LIN {X 0,Y 72.884,Z 397.402,A -85,B 0,C 180,E1 -28001.113,E2 -28001.113} C_VEL
LIN {X 0,Y 72.584,Z 397.443,A -85,B 0,C 180,E1 -28006.88,E2 -28006.88} C_VEL
LIN {X 0,Y 72.397,Z 397.459,A -85,B 0,C 180,E1 -28012.842,E2 -28012.842} C_VEL
LIN {X 0,Y 72.372,Z 397.464,A -85,B 0,C 180,E1 -28019.077,E2 -28019.077} C_VEL
LIN {X 0,Y 72.344,Z 397.474,A -85,B 0,C 180,E1 -28025.645,E2 -28025.645} C_VEL
LIN {X 0,Y 72.326,Z 397.475,A -85,B 0,C 180,E1 -28032.85,E2 -28032.85} C_VEL
LIN {X 0,Y 72.365,Z 397.469,A -85,B 0,C 180,E1 -28040.971,E2 -28040.971} C_VEL
LIN {X 0,Y 72.342,Z 397.472,A -85,B 0,C 180,E1 -28044.346,E2 -28044.346} C_VEL
LIN {X 0,Y 72.385,Z 397.468,A -85,B 0,C 180,E1 -28050.958,E2 -28050.958} C_VEL
LIN {X 0,Y 72.392,Z 397.461,A -85,B 0,C 180,E1 -28057.15,E2 -28057.15} C_VEL
LIN {X 0,Y 72.749,Z 397.413,A -85,B 0,C 180,E1 -28065.002,E2 -28065.002} C_VEL
LIN {X 0,Y 72.877,Z 397.407,A -85,B 0,C 180,E1 -28068.88,E2 -28068.88} C_VEL
LIN {X 0,Y 73.573,Z 397.317,A -85,B 0,C 180,E1 -28080.001,E2 -28080.001} C_VEL
LIN {X 0,Y 72.877,Z 397.398,A -85,B 0,C 180,E1 -28091.121,E2 -28091.121} C_VEL
LIN {X 0,Y 72.575,Z 397.443,A -85,B 0,C 180,E1 -28096.889,E2 -28096.889} C_VEL
LIN {X 0,Y 72.388,Z 397.467,A -85,B 0,C 180,E1 -28102.853,E2 -28102.853} C_VEL
LIN {X 0,Y 72.37,Z 397.461,A -85,B 0,C 180,E1 -28109.086,E2 -28109.086} C_VEL
LIN {X 0,Y 72.341,Z 397.469,A -85,B 0,C 180,E1 -28115.656,E2 -28115.656} C_VEL
LIN {X 0,Y 72.336,Z 397.474,A -85,B 0,C 180,E1 -28122.853,E2 -28122.853} C_VEL
LIN {X 0,Y 72.557,Z 397.447,A -85,B 0,C 180,E1 -28130.797,E2 -28130.797} C_VEL
LIN {X 0,Y 73.99,Z 397.266,A -85,B 0,C 180,E1 -28141.653,E2 -28141.653} C_VEL
LIN {X 0,Y 75.709,Z 408.16,A -85,B 0,C 180,E1 -28143.6,E2 -28143.6} C_VEL
LIN {X 0,Y 76.943,Z 433.067,A -85,B 0,C 180,E1 -28148.277,E2 -28148.277} C_VEL
LIN {X 0,Y 79.549,Z 458.898,A -85,B 0,C 180,E1 -28152.824,E2 -28152.824} C_VEL
LIN {X 0,Y 80.052,Z 501.083,A -85,B 0,C 180,E1 -28161.567,E2 -28161.567} C_VEL
LIN {X 0,Y 80.299,Z 512.942,A -85,B 0,C 180,E1 -28164.985,E2 -28164.985} C_VEL
LIN {X 0,Y 80.965,Z 525.078,A -85,B 0,C 180,E1 -28169.384,E2 -28169.384} C_VEL
LIN {X 0,Y 82.181,Z 537.066,A -85,B 0,C 180,E1 -28174.911,E2 -28174.911} C_VEL
LIN {X 0,Y 83.655,Z 545.69,A -85,B 0,C 180,E1 -28179.678,E2 -28179.678} C_VEL
LIN {X 0,Y 84.498,Z 549.412,A -85,B 0,C 180,E1 -28182.007,E2 -28182.007} C_VEL
LIN {X 0,Y 84.134,Z 553.13,A -85,B 0,C 180,E1 -28186.037,E2 -28186.037} C_VEL
LIN {X 0,Y 85.067,Z 561.406,A -85,B 0,C 180,E1 -28197.032,E2 -28197.032} C_VEL
LIN {X 0,Y 89.087,Z 567.646,A -85,B 0,C 180,E1 -28206.277,E2 -28206.277} C_VEL
LIN {X 0,Y 97.647,Z 574.029,A -85,B 0,C 180,E1 -28216.039,E2 -28216.039} C_VEL
LIN {X 0,Y 97.752,Z 573.898,A -85,B 0,C 180,E1 -28217.096,E2 -28217.096} C_VEL
LIN {X 0,Y 89.651,Z 565.539,A -85,B 0,C 180,E1 -28223.988,E2 -28223.988} C_VEL
LIN {X 0,Y 83.684,Z 555.645,A -85,B 0,C 180,E1 -28232.489,E2 -28232.489} C_VEL
LIN {X 0,Y 80.707,Z 546.935,A -85,B 0,C 180,E1 -28239.615,E2 -28239.615} C_VEL
LIN {X 0,Y 78.9,Z 536.529,A -85,B 0,C 180,E1 -28247.133,E2 -28247.133} C_VEL
LIN {X 0,Y 78.177,Z 528.616,A -85,B 0,C 180,E1 -28251.99,E2 -28251.99} C_VEL
LIN {X 0,Y 77.712,Z 518.041,A -85,B 0,C 180,E1 -28257.408,E2 -28257.408} C_VEL
LIN {X 0,Y 77.597,Z 505.51,A -85,B 0,C 180,E1 -28262.595,E2 -28262.595} C_VEL
LIN {X 0,Y 77.899,Z 492.74,A -85,B 0,C 180,E1 -28266.748,E2 -28266.748} C_VEL
LIN {X 0,Y 78.228,Z 475.491,A -85,B 0,C 180,E1 -28270.841,E2 -28270.841} C_VEL
LIN {X 0,Y 78.384,Z 437.977,A -85,B 0,C 180,E1 -28278.458,E2 -28278.458} C_VEL
LIN {X 0,Y 78.852,Z 421.185,A -85,B 0,C 180,E1 -28281.786,E2 -28281.786} C_VEL
LIN {X 0,Y 78.146,Z 418.606,A -85,B 0,C 180,E1 -28282.165,E2 -28282.165} C_VEL
LIN {X 0,Y 76.516,Z 414.995,A -85,B 0,C 180,E1 -28282.614,E2 -28282.614} C_VEL
LIN {X 0,Y 68.201,Z 404.386,A -85,B 0,C 180,E1 -28283.502,E2 -28283.502} C_VEL
LIN {X 0,Y 66.794,Z 400.744,A -85,B 0,C 180,E1 -28284.067,E2 -28284.067} C_VEL
LIN {X 0,Y 66.334,Z 398.209,A -85,B 0,C 180,E1 -28284.613,E2 -28284.613} C_VEL
LIN {X 0,Y 65.413,Z 398.327,A -85,B 0,C 180,E1 -28292.493,E2 -28292.493} C_VEL
LIN {X 0,Y 65.189,Z 398.356,A -85,B 0,C 180,E1 -28300.994,E2 -28300.994} C_VEL
LIN {X 0,Y 65.209,Z 398.353,A -85,B 0,C 180,E1 -28309.701,E2 -28309.701} C_VEL
LIN {X 0,Y 65.258,Z 398.346,A -85,B 0,C 180,E1 -28319.491,E2 -28319.491} C_VEL
LIN {X 0,Y 65.242,Z 398.358,A -85,B 0,C 180,E1 -28324.469,E2 -28324.469} C_VEL
LIN {X 0,Y 65.627,Z 398.307,A -85,B 0,C 180,E1 -28334.536,E2 -28334.536} C_VEL
LIN {X 0,Y 65.757,Z 398.285,A -85,B 0,C 180,E1 -28337.65,E2 -28337.65} C_VEL
LIN {X 0,Y 66.495,Z 398.203,A -85,B 0,C 180,E1 -28349.993,E2 -28349.993} C_VEL
LIN {X 0,Y 65.782,Z 398.282,A -85,B 0,C 180,E1 -28362.33,E2 -28362.33} C_VEL
LIN {X 0,Y 65.388,Z 398.339,A -85,B 0,C 180,E1 -28368.803,E2 -28368.803} C_VEL
LIN {X 0,Y 65.247,Z 398.357,A -85,B 0,C 180,E1 -28375.514,E2 -28375.514} C_VEL
LIN {X 0,Y 65.215,Z 398.356,A -85,B 0,C 180,E1 -28382.595,E2 -28382.595} C_VEL
LIN {X 0,Y 65.26,Z 398.349,A -85,B 0,C 180,E1 -28391.076,E2 -28391.076} C_VEL
LIN {X 0,Y 65.276,Z 398.347,A -85,B 0,C 180,E1 -28399.76,E2 -28399.76} C_VEL
LIN {X 0,Y 65.254,Z 398.353,A -85,B 0,C 180,E1 -28409.483,E2 -28409.483} C_VEL
LIN {X 0,Y 65.241,Z 398.351,A -85,B 0,C 180,E1 -28414.476,E2 -28414.476} C_VEL
LIN {X 0,Y 65.644,Z 398.298,A -85,B 0,C 180,E1 -28424.458,E2 -28424.458} C_VEL
LIN {X 0,Y 65.775,Z 398.29,A -85,B 0,C 180,E1 -28427.662,E2 -28427.662} C_VEL
LIN {X 0,Y 66.497,Z 398.198,A -85,B 0,C 180,E1 -28440.001,E2 -28440.001} C_VEL
LIN {X 0,Y 65.768,Z 398.285,A -85,B 0,C 180,E1 -28452.341,E2 -28452.341} C_VEL
LIN {X 0,Y 65.378,Z 398.333,A -85,B 0,C 180,E1 -28458.815,E2 -28458.815} C_VEL
LIN {X 0,Y 65.24,Z 398.357,A -85,B 0,C 180,E1 -28465.525,E2 -28465.525} C_VEL
LIN {X 0,Y 65.213,Z 398.362,A -85,B 0,C 180,E1 -28472.606,E2 -28472.606} C_VEL
LIN {X 0,Y 65.266,Z 398.355,A -85,B 0,C 180,E1 -28481.093,E2 -28481.093} C_VEL
LIN {X 0,Y 65.441,Z 398.334,A -85,B 0,C 180,E1 -28489.891,E2 -28489.891} C_VEL
LIN {X 0,Y 67.071,Z 398.126,A -85,B 0,C 180,E1 -28502.682,E2 -28502.682} C_VEL
LIN {X 0,Y 68.779,Z 409.161,A -85,B 0,C 180,E1 -28504.855,E2 -28504.855} C_VEL
LIN {X 0,Y 70.255,Z 434.542,A -85,B 0,C 180,E1 -28510.085,E2 -28510.085} C_VEL
LIN {X 0,Y 72.876,Z 458.865,A -85,B 0,C 180,E1 -28514.729,E2 -28514.729} C_VEL
LIN {X 0,Y 73.916,Z 500.644,A -85,B 0,C 180,E1 -28524.208,E2 -28524.208} C_VEL
LIN {X 0,Y 74.379,Z 512.529,A -85,B 0,C 180,E1 -28527.976,E2 -28527.976} C_VEL
LIN {X 0,Y 75.35,Z 524.438,A -85,B 0,C 180,E1 -28532.679,E2 -28532.679} C_VEL
LIN {X 0,Y 76.78,Z 535.088,A -85,B 0,C 180,E1 -28537.898,E2 -28537.898} C_VEL
LIN {X 0,Y 78.569,Z 543.731,A -85,B 0,C 180,E1 -28542.928,E2 -28542.928} C_VEL
LIN {X 0,Y 79.079,Z 545.678,A -85,B 0,C 180,E1 -28544.152,E2 -28544.152} C_VEL
LIN {X 0,Y 79.134,Z 547.078,A -85,B 0,C 180,E1 -28545.458,E2 -28545.458} C_VEL
LIN {X 0,Y 79.462,Z 555.198,A -85,B 0,C 180,E1 -28556.252,E2 -28556.252} C_VEL
LIN {X 0,Y 83.073,Z 562.054,A -85,B 0,C 180,E1 -28566.32,E2 -28566.32} C_VEL
LIN {X 0,Y 89.595,Z 567.905,A -85,B 0,C 180,E1 -28575.091,E2 -28575.091} C_VEL
LIN {X 0,Y 89.992,Z 567.977,A -85,B 0,C 180,E1 -28576.643,E2 -28576.643} C_VEL
LIN {X 0,Y 81.965,Z 558.323,A -85,B 0,C 180,E1 -28584.635,E2 -28584.635} C_VEL
LIN {X 0,Y 77.144,Z 548.736,A -85,B 0,C 180,E1 -28592.901,E2 -28592.901} C_VEL
LIN {X 0,Y 74.209,Z 538.508,A -85,B 0,C 180,E1 -28600.929,E2 -28600.929} C_VEL
LIN {X 0,Y 72.923,Z 529.145,A -85,B 0,C 180,E1 -28607.475,E2 -28607.475} C_VEL
LIN {X 0,Y 71.984,Z 518.076,A -85,B 0,C 180,E1 -28613.693,E2 -28613.693} C_VEL
LIN {X 0,Y 71.557,Z 506.061,A -85,B 0,C 180,E1 -28619.165,E2 -28619.165} C_VEL
LIN {X 0,Y 71.591,Z 494.153,A -85,B 0,C 180,E1 -28623.517,E2 -28623.517} C_VEL
LIN {X 0,Y 71.771,Z 478.582,A -85,B 0,C 180,E1 -28627.737,E2 -28627.737} C_VEL
LIN {X 0,Y 71.636,Z 448.711,A -85,B 0,C 180,E1 -28634.56,E2 -28634.56} C_VEL
LIN {X 0,Y 71.869,Z 421.52,A -85,B 0,C 180,E1 -28640.517,E2 -28640.517} C_VEL
LIN {X 0,Y 67.195,Z 402.969,A -85,B 0,C 180,E1 -28643.639,E2 -28643.639} C_VEL
LIN {X 0,Y 66.794,Z 400.744,A -85,B 0,C 180,E1 -28644.067,E2 -28644.067} C_VEL
LIN {X 0,Y 66.151,Z 399.397,A -85,B 0,C 180,E1 -28644.879,E2 -28644.879} C_VEL
LIN {X 0,Y 64.817,Z 398.602,A -85,B 0,C 180,E1 -28646.815,E2 -28646.815} C_VEL
LIN {X 0,Y 60.938,Z 398.887,A -85,B 0,C 180,E1 -28654.521,E2 -28654.521} C_VEL
LIN {X 0,Y 58.572,Z 399.406,A -85,B 0,C 180,E1 -28663.21,E2 -28663.21} C_VEL
LIN {X 0,Y 58.022,Z 399.251,A -85,B 0,C 180,E1 -28672.443,E2 -28672.443} C_VEL
LIN {X 0,Y 58.163,Z 399.232,A -85,B 0,C 180,E1 -28677.76,E2 -28677.76} C_VEL
LIN {X 0,Y 58.155,Z 399.234,A -85,B 0,C 180,E1 -28681.083,E2 -28681.083} C_VEL
LIN {X 0,Y 58.519,Z 399.194,A -85,B 0,C 180,E1 -28693.899,E2 -28693.899} C_VEL
LIN {X 0,Y 58.802,Z 399.157,A -85,B 0,C 180,E1 -28703.128,E2 -28703.128} C_VEL
LIN {X 0,Y 59.386,Z 399.088,A -85,B 0,C 180,E1 -28709.992,E2 -28709.992} C_VEL
LIN {X 0,Y 58.824,Z 399.154,A -85,B 0,C 180,E1 -28716.854,E2 -28716.854} C_VEL
LIN {X 0,Y 58.535,Z 399.192,A -85,B 0,C 180,E1 -28726.157,E2 -28726.157} C_VEL
LIN {X 0,Y 58.155,Z 399.234,A -85,B 0,C 180,E1 -28738.898,E2 -28738.898} C_VEL
LIN {X 0,Y 58.08,Z 399.246,A -85,B 0,C 180,E1 -28747.221,E2 -28747.221} C_VEL
LIN {X 0,Y 58.102,Z 399.241,A -85,B 0,C 180,E1 -28756.519,E2 -28756.519} C_VEL
LIN {X 0,Y 58.078,Z 399.251,A -85,B 0,C 180,E1 -28762.769,E2 -28762.769} C_VEL
LIN {X 0,Y 58.152,Z 399.241,A -85,B 0,C 180,E1 -28771.091,E2 -28771.091} C_VEL
LIN {X 0,Y 58.53,Z 399.185,A -85,B 0,C 180,E1 -28783.834,E2 -28783.834} C_VEL
LIN {X 0,Y 58.816,Z 399.149,A -85,B 0,C 180,E1 -28793.138,E2 -28793.138} C_VEL
LIN {X 0,Y 59.389,Z 399.083,A -85,B 0,C 180,E1 -28800.001,E2 -28800.001} C_VEL
LIN {X 0,Y 58.816,Z 399.159,A -85,B 0,C 180,E1 -28806.864,E2 -28806.864} C_VEL
LIN {X 0,Y 58.518,Z 399.195,A -85,B 0,C 180,E1 -28816.128,E2 -28816.128} C_VEL
LIN {X 0,Y 58.15,Z 399.232,A -85,B 0,C 180,E1 -28828.911,E2 -28828.911} C_VEL
LIN {X 0,Y 58.081,Z 399.24,A -85,B 0,C 180,E1 -28837.231,E2 -28837.231} C_VEL
LIN {X 0,Y 58.186,Z 399.227,A -85,B 0,C 180,E1 -28846.446,E2 -28846.446} C_VEL
LIN {X 0,Y 58.897,Z 399.14,A -85,B 0,C 180,E1 -28856.648,E2 -28856.648} C_VEL
LIN {X 0,Y 60.22,Z 398.977,A -85,B 0,C 180,E1 -28864.088,E2 -28864.088} C_VEL
LIN {X 0,Y 61.903,Z 409.857,A -85,B 0,C 180,E1 -28866.433,E2 -28866.433} C_VEL
LIN {X 0,Y 63.446,Z 433.388,A -85,B 0,C 180,E1 -28871.799,E2 -28871.799} C_VEL
LIN {X 0,Y 66.355,Z 458.968,A -85,B 0,C 180,E1 -28877.137,E2 -28877.137} C_VEL
LIN {X 0,Y 68.011,Z 500.189,A -85,B 0,C 180,E1 -28887.416,E2 -28887.416} C_VEL
LIN {X 0,Y 68.741,Z 511.901,A -85,B 0,C 180,E1 -28891.471,E2 -28891.471} C_VEL
LIN {X 0,Y 70.075,Z 523.639,A -85,B 0,C 180,E1 -28896.485,E2 -28896.485} C_VEL
LIN {X 0,Y 72.148,Z 535.102,A -85,B 0,C 180,E1 -28902.523,E2 -28902.523} C_VEL
LIN {X 0,Y 73.814,Z 541.67,A -85,B 0,C 180,E1 -28906.603,E2 -28906.603} C_VEL
LIN {X 0,Y 74.056,Z 543.545,A -85,B 0,C 180,E1 -28908.372,E2 -28908.372} C_VEL
LIN {X 0,Y 75.288,Z 552.281,A -85,B 0,C 180,E1 -28920.557,E2 -28920.557} C_VEL
LIN {X 0,Y 80.097,Z 559.341,A -85,B 0,C 180,E1 -28931.16,E2 -28931.16} C_VEL
LIN {X 0,Y 82.912,Z 561.871,A -85,B 0,C 180,E1 -28934.893,E2 -28934.893} C_VEL
LIN {X 0,Y 81.955,Z 560.671,A -85,B 0,C 180,E1 -28936.682,E2 -28936.682} C_VEL
LIN {X 0,Y 74.644,Z 550.167,A -85,B 0,C 180,E1 -28945.602,E2 -28945.602} C_VEL
LIN {X 0,Y 70.806,Z 541.09,A -85,B 0,C 180,E1 -28953.306,E2 -28953.306} C_VEL
LIN {X 0,Y 68.092,Z 529.146,A -85,B 0,C 180,E1 -28962.428,E2 -28962.428} C_VEL
LIN {X 0,Y 66.732,Z 518.591,A -85,B 0,C 180,E1 -28968.995,E2 -28968.995} C_VEL
LIN {X 0,Y 65.901,Z 506.552,A -85,B 0,C 180,E1 -28975.065,E2 -28975.065} C_VEL
LIN {X 0,Y 65.609,Z 493.245,A -85,B 0,C 180,E1 -28980.383,E2 -28980.383} C_VEL
LIN {X 0,Y 65.57,Z 476.574,A -85,B 0,C 180,E1 -28985.284,E2 -28985.284} C_VEL
LIN {X 0,Y 64.904,Z 442.925,A -85,B 0,C 180,E1 -28993.731,E2 -28993.731} C_VEL
LIN {X 0,Y 65.039,Z 422.11,A -85,B 0,C 180,E1 -28998.813,E2 -28998.813} C_VEL
LIN {X 0,Y 60.331,Z 403.573,A -85,B 0,C 180,E1 -29002.159,E2 -29002.159} C_VEL
LIN {X 0,Y 59.457,Z 399.066,A -85,B 0,C 180,E1 -29003.193,E2 -29003.193} C_VEL
LIN {X 0,Y 58.104,Z 399.247,A -85,B 0,C 180,E1 -29017.212,E2 -29017.212} C_VEL
LIN {X 0,Y 58.018,Z 399.258,A -85,B 0,C 180,E1 -29026.618,E2 -29026.618} C_VEL
LIN {X 0,Y 58.022,Z 399.251,A -85,B 0,C 180,E1 -29032.443,E2 -29032.443} C_VEL
LIN {X 0,Y 57.853,Z 399.288,A -85,B 0,C 180,E1 -29036.305,E2 -29036.305} C_VEL
LIN {X 0,Y 56.621,Z 399.45,A -85,B 0,C 180,E1 -29042.093,E2 -29042.093} C_VEL
LIN {X 0,Y 54.829,Z 399.669,A -85,B 0,C 180,E1 -29047.958,E2 -29047.958} C_VEL
LIN {X 0,Y 51.867,Z 400.025,A -85,B 0,C 180,E1 -29061.019,E2 -29061.019} C_VEL
LIN {X 0,Y 51.817,Z 400.015,A -85,B 0,C 180,E1 -29065.612,E2 -29065.612} C_VEL
LIN {X 0,Y 52.269,Z 399.975,A -85,B 0,C 180,E1 -29069.991,E2 -29069.991} C_VEL
LIN {X 0,Y 51.7,Z 400.044,A -85,B 0,C 180,E1 -29077.804,E2 -29077.804} C_VEL
LIN {X 0,Y 51.401,Z 400.082,A -85,B 0,C 180,E1 -29086.847,E2 -29086.847} C_VEL
LIN {X 0,Y 51.027,Z 400.124,A -85,B 0,C 180,E1 -29094.395,E2 -29094.395} C_VEL
LIN {X 0,Y 51.053,Z 400.125,A -85,B 0,C 180,E1 -29104.315,E2 -29104.315} C_VEL
LIN {X 0,Y 51.067,Z 400.124,A -85,B 0,C 180,E1 -29113.468,E2 -29113.468} C_VEL
LIN {X 0,Y 51.067,Z 400.117,A -85,B 0,C 180,E1 -29116.52,E2 -29116.52} C_VEL
LIN {X 0,Y 51.074,Z 400.113,A -85,B 0,C 180,E1 -29126.605,E2 -29126.605} C_VEL
LIN {X 0,Y 51.023,Z 400.119,A -85,B 0,C 180,E1 -29135.593,E2 -29135.593} C_VEL
LIN {X 0,Y 51.474,Z 400.063,A -85,B 0,C 180,E1 -29144.154,E2 -29144.154} C_VEL
LIN {X 0,Y 51.692,Z 400.037,A -85,B 0,C 180,E1 -29152.187,E2 -29152.187} C_VEL
LIN {X 0,Y 52.274,Z 399.968,A -85,B 0,C 180,E1 -29160.001,E2 -29160.001} C_VEL
LIN {X 0,Y 51.69,Z 400.045,A -85,B 0,C 180,E1 -29167.815,E2 -29167.815} C_VEL
LIN {X 0,Y 51.386,Z 400.082,A -85,B 0,C 180,E1 -29176.822,E2 -29176.822} C_VEL
LIN {X 0,Y 51.021,Z 400.13,A -85,B 0,C 180,E1 -29184.409,E2 -29184.409} C_VEL
LIN {X 0,Y 51.052,Z 400.123,A -85,B 0,C 180,E1 -29194.329,E2 -29194.329} C_VEL
LIN {X 0,Y 51.168,Z 400.101,A -85,B 0,C 180,E1 -29206.639,E2 -29206.639} C_VEL
LIN {X 0,Y 52.619,Z 399.925,A -85,B 0,C 180,E1 -29222.144,E2 -29222.144} C_VEL
LIN {X 0,Y 53.445,Z 399.843,A -85,B 0,C 180,E1 -29226.07,E2 -29226.07} C_VEL
LIN {X 0,Y 55.057,Z 409.615,A -85,B 0,C 180,E1 -29228.28,E2 -29228.28} C_VEL
LIN {X 0,Y 57.04,Z 435.1,A -85,B 0,C 180,E1 -29234.716,E2 -29234.716} C_VEL
LIN {X 0,Y 60.017,Z 458.109,A -85,B 0,C 180,E1 -29239.891,E2 -29239.891} C_VEL
LIN {X 0,Y 62.423,Z 499.448,A -85,B 0,C 180,E1 -29251.218,E2 -29251.218} C_VEL
LIN {X 0,Y 63.485,Z 511.276,A -85,B 0,C 180,E1 -29255.647,E2 -29255.647} C_VEL
LIN {X 0,Y 64.967,Z 521.199,A -85,B 0,C 180,E1 -29260.132,E2 -29260.132} C_VEL
LIN {X 0,Y 67.209,Z 531.883,A -85,B 0,C 180,E1 -29265.937,E2 -29265.937} C_VEL
LIN {X 0,Y 69.019,Z 538.028,A -85,B 0,C 180,E1 -29269.767,E2 -29269.767} C_VEL
LIN {X 0,Y 69.27,Z 539.215,A -85,B 0,C 180,E1 -29270.828,E2 -29270.828} C_VEL
LIN {X 0,Y 71.033,Z 547.999,A -85,B 0,C 180,E1 -29283.485,E2 -29283.485} C_VEL
LIN {X 0,Y 76.015,Z 554.814,A -85,B 0,C 180,E1 -29293.837,E2 -29293.837} C_VEL
LIN {X 0,Y 75.472,Z 553.984,A -85,B 0,C 180,E1 -29295.7,E2 -29295.7} C_VEL
LIN {X 0,Y 68.382,Z 542.524,A -85,B 0,C 180,E1 -29305.575,E2 -29305.575} C_VEL
LIN {X 0,Y 64.548,Z 532.018,A -85,B 0,C 180,E1 -29314.181,E2 -29314.181} C_VEL
LIN {X 0,Y 62.84,Z 523.725,A -85,B 0,C 180,E1 -29320.395,E2 -29320.395} C_VEL
LIN {X 0,Y 61.304,Z 513.354,A -85,B 0,C 180,E1 -29326.744,E2 -29326.744} C_VEL
LIN {X 0,Y 60.319,Z 502.043,A -85,B 0,C 180,E1 -29332.467,E2 -29332.467} C_VEL
LIN {X 0,Y 59.891,Z 489.793,A -85,B 0,C 180,E1 -29337.477,E2 -29337.477} C_VEL
LIN {X 0,Y 59.468,Z 472.762,A -85,B 0,C 180,E1 -29342.751,E2 -29342.751} C_VEL
LIN {X 0,Y 58.275,Z 438.279,A -85,B 0,C 180,E1 -29352.297,E2 -29352.297} C_VEL
LIN {X 0,Y 58.235,Z 422.432,A -85,B 0,C 180,E1 -29356.652,E2 -29356.652} C_VEL
LIN {X 0,Y 53.572,Z 404.309,A -85,B 0,C 180,E1 -29360.124,E2 -29360.124} C_VEL
LIN {X 0,Y 52.653,Z 399.921,A -85,B 0,C 180,E1 -29361.338,E2 -29361.338} C_VEL
LIN {X 0,Y 51.143,Z 400.106,A -85,B 0,C 180,E1 -29374.446,E2 -29374.446} C_VEL
LIN {X 0,Y 50.985,Z 400.134,A -85,B 0,C 180,E1 -29386.419,E2 -29386.419} C_VEL
LIN {X 0,Y 51.055,Z 400.122,A -85,B 0,C 180,E1 -29396.58,E2 -29396.58} C_VEL
LIN {X 0,Y 51.026,Z 400.125,A -85,B 0,C 180,E1 -29405.584,E2 -29405.584} C_VEL
LIN {X 0,Y 51.46,Z 400.072,A -85,B 0,C 180,E1 -29414.139,E2 -29414.139} C_VEL
LIN {X 0,Y 51.817,Z 400.015,A -85,B 0,C 180,E1 -29425.612,E2 -29425.612} C_VEL
LIN {X 0,Y 51.492,Z 400.071,A -85,B 0,C 180,E1 -29429.149,E2 -29429.149} C_VEL
LIN {X 0,Y 49.798,Z 400.291,A -85,B 0,C 180,E1 -29433.965,E2 -29433.965} C_VEL
LIN {X 0,Y 44.332,Z 400.965,A -85,B 0,C 180,E1 -29447.752,E2 -29447.752} C_VEL
LIN {X 0,Y 44.096,Z 400.983,A -85,B 0,C 180,E1 -29449.551,E2 -29449.551} C_VEL
LIN {X 0,Y 43.856,Z 401.015,A -85,B 0,C 180,E1 -29458.722,E2 -29458.722} C_VEL
LIN {X 0,Y 43.873,Z 401.01,A -85,B 0,C 180,E1 -29469.835,E2 -29469.835} C_VEL
LIN {X 0,Y 43.907,Z 401.016,A -85,B 0,C 180,E1 -29483.142,E2 -29483.142} C_VEL
LIN {X 0,Y 43.853,Z 401.023,A -85,B 0,C 180,E1 -29491.264,E2 -29491.264} C_VEL
LIN {X 0,Y 44.25,Z 400.967,A -85,B 0,C 180,E1 -29502.317,E2 -29502.317} C_VEL
LIN {X 0,Y 44.544,Z 400.931,A -85,B 0,C 180,E1 -29510.923,E2 -29510.923} C_VEL
LIN {X 0,Y 45.149,Z 400.855,A -85,B 0,C 180,E1 -29520.001,E2 -29520.001} C_VEL
LIN {X 0,Y 44.539,Z 400.93,A -85,B 0,C 180,E1 -29529.08,E2 -29529.08} C_VEL
LIN {X 0,Y 44.15,Z 400.976,A -85,B 0,C 180,E1 -29538.566,E2 -29538.566} C_VEL
LIN {X 0,Y 43.853,Z 401.012,A -85,B 0,C 180,E1 -29548.738,E2 -29548.738} C_VEL
LIN {X 0,Y 43.896,Z 401.012,A -85,B 0,C 180,E1 -29559.825,E2 -29559.825} C_VEL
LIN {X 0,Y 44.308,Z 400.96,A -85,B 0,C 180,E1 -29572.477,E2 -29572.477} C_VEL
LIN {X 0,Y 46.765,Z 400.659,A -85,B 0,C 180,E1 -29588.607,E2 -29588.607} C_VEL
LIN {X 0,Y 48.333,Z 409.803,A -85,B 0,C 180,E1 -29590.958,E2 -29590.958} C_VEL
LIN {X 0,Y 50.773,Z 435.813,A -85,B 0,C 180,E1 -29598.24,E2 -29598.24} C_VEL
LIN {X 0,Y 53.923,Z 458.116,A -85,B 0,C 180,E1 -29603.695,E2 -29603.695} C_VEL
LIN {X 0,Y 57.212,Z 498.454,A -85,B 0,C 180,E1 -29615.735,E2 -29615.735} C_VEL
LIN {X 0,Y 58.633,Z 510.019,A -85,B 0,C 180,E1 -29620.366,E2 -29620.366} C_VEL
LIN {X 0,Y 60.601,Z 520.498,A -85,B 0,C 180,E1 -29625.396,E2 -29625.396} C_VEL
LIN {X 0,Y 63.706,Z 531.833,A -85,B 0,C 180,E1 -29631.885,E2 -29631.885} C_VEL
LIN {X 0,Y 64.779,Z 534.938,A -85,B 0,C 180,E1 -29633.908,E2 -29633.908} C_VEL
LIN {X 0,Y 67.404,Z 544.014,A -85,B 0,C 180,E1 -29647.44,E2 -29647.44} C_VEL
LIN {X 0,Y 69.896,Z 547.579,A -85,B 0,C 180,E1 -29652.96,E2 -29652.96} C_VEL
LIN {X 0,Y 69.317,Z 546.679,A -85,B 0,C 180,E1 -29654.786,E2 -29654.786} C_VEL
LIN {X 0,Y 63.264,Z 536.075,A -85,B 0,C 180,E1 -29663.846,E2 -29663.846} C_VEL
LIN {X 0,Y 59.175,Z 524.061,A -85,B 0,C 180,E1 -29673.552,E2 -29673.552} C_VEL
LIN {X 0,Y 57.094,Z 514.187,A -85,B 0,C 180,E1 -29680.213,E2 -29680.213} C_VEL
LIN {X 0,Y 55.612,Z 503.425,A -85,B 0,C 180,E1 -29686.292,E2 -29686.292} C_VEL
LIN {X 0,Y 54.634,Z 490.582,A -85,B 0,C 180,E1 -29692.144,E2 -29692.144} C_VEL
LIN {X 0,Y 53.818,Z 473.473,A -85,B 0,C 180,E1 -29698.128,E2 -29698.128} C_VEL
LIN {X 0,Y 52.002,Z 440.349,A -85,B 0,C 180,E1 -29708.347,E2 -29708.347} C_VEL
LIN {X 0,Y 51.519,Z 422.361,A -85,B 0,C 180,E1 -29713.897,E2 -29713.897} C_VEL
LIN {X 0,Y 46.851,Z 404.631,A -85,B 0,C 180,E1 -29717.457,E2 -29717.457} C_VEL
LIN {X 0,Y 46.049,Z 400.748,A -85,B 0,C 180,E1 -29718.505,E2 -29718.505} C_VEL
LIN {X 0,Y 43.932,Z 401.013,A -85,B 0,C 180,E1 -29736.865,E2 -29736.865} C_VEL
LIN {X 0,Y 43.806,Z 401.018,A -85,B 0,C 180,E1 -29750.065,E2 -29750.065} C_VEL
LIN {X 0,Y 43.847,Z 401.016,A -85,B 0,C 180,E1 -29761.247,E2 -29761.247} C_VEL
LIN {X 0,Y 44.231,Z 400.976,A -85,B 0,C 180,E1 -29772.43,E2 -29772.43} C_VEL
LIN {X 0,Y 44.531,Z 400.938,A -85,B 0,C 180,E1 -29780.909,E2 -29780.909} C_VEL
LIN {X 0,Y 45.143,Z 400.862,A -85,B 0,C 180,E1 -29789.99,E2 -29789.99} C_VEL
LIN {X 0,Y 44.551,Z 400.936,A -85,B 0,C 180,E1 -29799.066,E2 -29799.066} C_VEL
LIN {X 0,Y 44.096,Z 400.983,A -85,B 0,C 180,E1 -29809.551,E2 -29809.551} C_VEL
LIN {X 0,Y 43.388,Z 401.076,A -85,B 0,C 180,E1 -29814.623,E2 -29814.623} C_VEL
LIN {X 0,Y 41.673,Z 401.291,A -85,B 0,C 180,E1 -29822.278,E2 -29822.278} C_VEL
LIN {X 0,Y 39.664,Z 401.534,A -85,B 0,C 180,E1 -29830.224,E2 -29830.224} C_VEL
LIN {X 0,Y 36.682,Z 401.889,A -85,B 0,C 180,E1 -29854.884,E2 -29854.884} C_VEL
LIN {X 0,Y 37.074,Z 401.864,A -85,B 0,C 180,E1 -29861.37,E2 -29861.37} C_VEL
LIN {X 0,Y 37.342,Z 401.834,A -85,B 0,C 180,E1 -29869.153,E2 -29869.153} C_VEL
LIN {X 0,Y 38.007,Z 401.743,A -85,B 0,C 180,E1 -29880.001,E2 -29880.001} C_VEL
LIN {X 0,Y 37.331,Z 401.824,A -85,B 0,C 180,E1 -29890.853,E2 -29890.853} C_VEL
LIN {X 0,Y 37.052,Z 401.86,A -85,B 0,C 180,E1 -29898.527,E2 -29898.527} C_VEL
LIN {X 0,Y 36.757,Z 401.899,A -85,B 0,C 180,E1 -29915.003,E2 -29915.003} C_VEL
LIN {X 0,Y 36.836,Z 401.892,A -85,B 0,C 180,E1 -29920.275,E2 -29920.275} C_VEL
LIN {X 0,Y 37.44,Z 401.811,A -85,B 0,C 180,E1 -29935.743,E2 -29935.743} C_VEL
LIN {X 0,Y 40.252,Z 401.461,A -85,B 0,C 180,E1 -29952.141,E2 -29952.141} C_VEL
LIN {X 0,Y 41.826,Z 409.981,A -85,B 0,C 180,E1 -29954.619,E2 -29954.619} C_VEL
LIN {X 0,Y 44.866,Z 436.866,A -85,B 0,C 180,E1 -29962.981,E2 -29962.981} C_VEL
LIN {X 0,Y 48.206,Z 457.818,A -85,B 0,C 180,E1 -29968.443,E2 -29968.443} C_VEL
LIN {X 0,Y 52.403,Z 496.818,A -85,B 0,C 180,E1 -29980.969,E2 -29980.969} C_VEL
LIN {X 0,Y 53.969,Z 506.894,A -85,B 0,C 180,E1 -29985.105,E2 -29985.105} C_VEL
LIN {X 0,Y 56.657,Z 518.761,A -85,B 0,C 180,E1 -29990.902,E2 -29990.902} C_VEL
LIN {X 0,Y 60.035,Z 529.169,A -85,B 0,C 180,E1 -29996.926,E2 -29996.926} C_VEL
LIN {X 0,Y 60.488,Z 530.385,A -85,B 0,C 180,E1 -29997.703,E2 -29997.703} C_VEL
LIN {X 0,Y 60.902,Z 531.883,A -85,B 0,C 180,E1 -29999.38,E2 -29999.38} C_VEL
LIN {X 0,Y 63.997,Z 539.515,A -85,B 0,C 180,E1 -30011.226,E2 -30011.226} C_VEL
LIN {X 0,Y 62.912,Z 537.776,A -85,B 0,C 180,E1 -30014.564,E2 -30014.564} C_VEL
LIN {X 0,Y 58.747,Z 529.93,A -85,B 0,C 180,E1 -30021.089,E2 -30021.089} C_VEL
LIN {X 0,Y 55.091,Z 519.736,A -85,B 0,C 180,E1 -30029.316,E2 -30029.316} C_VEL
LIN {X 0,Y 52.517,Z 509.133,A -85,B 0,C 180,E1 -30036.329,E2 -30036.329} C_VEL
LIN {X 0,Y 50.652,Z 497.279,A -85,B 0,C 180,E1 -30042.851,E2 -30042.851} C_VEL
LIN {X 0,Y 49.518,Z 484.586,A -85,B 0,C 180,E1 -30048.486,E2 -30048.486} C_VEL
LIN {X 0,Y 47.903,Z 465.058,A -85,B 0,C 180,E1 -30055.529,E2 -30055.529} C_VEL
LIN {X 0,Y 45.18,Z 422.904,A -85,B 0,C 180,E1 -30070.08,E2 -30070.08} C_VEL
LIN {X 0,Y 40.651,Z 406.325,A -85,B 0,C 180,E1 -30073.429,E2 -30073.429} C_VEL
LIN {X 0,Y 39.554,Z 401.548,A -85,B 0,C 180,E1 -30074.862,E2 -30074.862} C_VEL
LIN {X 0,Y 36.923,Z 401.877,A -85,B 0,C 180,E1 -30094.82,E2 -30094.82} C_VEL
LIN {X 0,Y 36.769,Z 401.896,A -85,B 0,C 180,E1 -30100.114,E2 -30100.114} C_VEL
LIN {X 0,Y 36.732,Z 401.899,A -85,B 0,C 180,E1 -30109.935,E2 -30109.935} C_VEL
LIN {X 0,Y 36.727,Z 401.911,A -85,B 0,C 180,E1 -30114.95,E2 -30114.95} C_VEL
LIN {X 0,Y 37.057,Z 401.866,A -85,B 0,C 180,E1 -30131.485,E2 -30131.485} C_VEL
LIN {X 0,Y 37.329,Z 401.828,A -85,B 0,C 180,E1 -30139.135,E2 -30139.135} C_VEL
LIN {X 0,Y 38.001,Z 401.752,A -85,B 0,C 180,E1 -30149.988,E2 -30149.988} C_VEL
LIN {X 0,Y 37.348,Z 401.826,A -85,B 0,C 180,E1 -30160.833,E2 -30160.833} C_VEL
LIN {X 0,Y 37.079,Z 401.863,A -85,B 0,C 180,E1 -30168.616,E2 -30168.616} C_VEL
LIN {X 0,Y 36.757,Z 401.907,A -85,B 0,C 180,E1 -30184.986,E2 -30184.986} C_VEL
LIN {X 0,Y 36.782,Z 401.893,A -85,B 0,C 180,E1 -30190.158,E2 -30190.158} C_VEL
LIN {X 0,Y 36.781,Z 401.894,A -85,B 0,C 180,E1 -30199.826,E2 -30199.826} C_VEL
LIN {X 0,Y 36.765,Z 401.898,A -85,B 0,C 180,E1 -30205.008,E2 -30205.008} C_VEL
LIN {X 0,Y 36.682,Z 401.889,A -85,B 0,C 180,E1 -30214.884,E2 -30214.884} C_VEL
LIN {X 0,Y 36.394,Z 401.952,A -85,B 0,C 180,E1 -30219.899,E2 -30219.899} C_VEL
LIN {X 0,Y 34.873,Z 402.146,A -85,B 0,C 180,E1 -30226.856,E2 -30226.856} C_VEL
LIN {X 0,Y 30.12,Z 402.6,A -85,B 0,C 180,E1 -30250.355,E2 -30250.355} C_VEL
LIN {X 0,Y 29.869,Z 402.635,A -85,B 0,C 180,E1 -30259.797,E2 -30259.797} C_VEL
LIN {X 0,Y 29.545,Z 402.666,A -85,B 0,C 180,E1 -30268.409,E2 -30268.409} C_VEL
LIN {X 0,Y 29.768,Z 402.646,A -85,B 0,C 180,E1 -30285.097,E2 -30285.097} C_VEL
LIN {X 0,Y 32.449,Z 402.393,A -85,B 0,C 180,E1 -30311.057,E2 -30311.057} C_VEL
LIN {X 0,Y 34.097,Z 402.432,A -85,B 0,C 180,E1 -30317.449,E2 -30317.449} C_VEL
LIN {X 0,Y 35.664,Z 410.432,A -85,B 0,C 180,E1 -30319.845,E2 -30319.845} C_VEL
LIN {X 0,Y 38.977,Z 435.166,A -85,B 0,C 180,E1 -30328.398,E2 -30328.398} C_VEL
LIN {X 0,Y 42.952,Z 457.162,A -85,B 0,C 180,E1 -30334.391,E2 -30334.391} C_VEL
LIN {X 0,Y 48.578,Z 497.018,A -85,B 0,C 180,E1 -30347.915,E2 -30347.915} C_VEL
LIN {X 0,Y 51.164,Z 509.167,A -85,B 0,C 180,E1 -30353.27,E2 -30353.27} C_VEL
LIN {X 0,Y 54.467,Z 520.136,A -85,B 0,C 180,E1 -30358.948,E2 -30358.948} C_VEL
LIN {X 0,Y 56.972,Z 526.471,A -85,B 0,C 180,E1 -30362.614,E2 -30362.614} C_VEL
LIN {X 0,Y 57.312,Z 527.337,A -85,B 0,C 180,E1 -30363.423,E2 -30363.423} C_VEL
LIN {X 0,Y 58.698,Z 531.027,A -85,B 0,C 180,E1 -30369.329,E2 -30369.329} C_VEL
LIN {X 0,Y 58.784,Z 531.304,A -85,B 0,C 180,E1 -30371.648,E2 -30371.648} C_VEL
LIN {X 0,Y 53.064,Z 519.625,A -85,B 0,C 180,E1 -30381.014,E2 -30381.014} C_VEL
LIN {X 0,Y 50.606,Z 512.35,A -85,B 0,C 180,E1 -30386.253,E2 -30386.253} C_VEL
LIN {X 0,Y 48.001,Z 501.953,A -85,B 0,C 180,E1 -30392.652,E2 -30392.652} C_VEL
LIN {X 0,Y 45.861,Z 488.552,A -85,B 0,C 180,E1 -30399.537,E2 -30399.537} C_VEL
LIN {X 0,Y 43.84,Z 471.564,A -85,B 0,C 180,E1 -30406.414,E2 -30406.414} C_VEL
LIN {X 0,Y 40.05,Z 437.012,A -85,B 0,C 180,E1 -30419.37,E2 -30419.37} C_VEL
LIN {X 0,Y 38.997,Z 422.936,A -85,B 0,C 180,E1 -30424.957,E2 -30424.957} C_VEL
LIN {X 0,Y 34.341,Z 406.278,A -85,B 0,C 180,E1 -30428.265,E2 -30428.265} C_VEL
LIN {X 0,Y 33.349,Z 402.311,A -85,B 0,C 180,E1 -30429.563,E2 -30429.563} C_VEL
LIN {X 0,Y 30.23,Z 402.606,A -85,B 0,C 180,E1 -30447.706,E2 -30447.706} C_VEL
LIN {X 0,Y 29.586,Z 402.666,A -85,B 0,C 180,E1 -30465.448,E2 -30465.448} C_VEL
LIN {X 0,Y 29.498,Z 402.672,A -85,B 0,C 180,E1 -30481.525,E2 -30481.525} C_VEL
LIN {X 0,Y 29.866,Z 402.638,A -85,B 0,C 180,E1 -30490.263,E2 -30490.263} C_VEL
LIN {X 0,Y 30.107,Z 402.614,A -85,B 0,C 180,E1 -30496.485,E2 -30496.485} C_VEL
LIN {X 0,Y 30.818,Z 402.551,A -85,B 0,C 180,E1 -30509.985,E2 -30509.985} C_VEL
LIN {X 0,Y 30.126,Z 402.612,A -85,B 0,C 180,E1 -30523.475,E2 -30523.475} C_VEL
LIN {X 0,Y 29.89,Z 402.635,A -85,B 0,C 180,E1 -30529.867,E2 -30529.867} C_VEL
LIN {X 0,Y 29.554,Z 402.667,A -85,B 0,C 180,E1 -30538.381,E2 -30538.381} C_VEL
LIN {X 0,Y 29.596,Z 402.664,A -85,B 0,C 180,E1 -30555.406,E2 -30555.406} C_VEL
LIN {X 0,Y 29.555,Z 402.668,A -85,B 0,C 180,E1 -30571.604,E2 -30571.604} C_VEL
LIN {X 0,Y 29.885,Z 402.637,A -85,B 0,C 180,E1 -30580.115,E2 -30580.115} C_VEL
LIN {X 0,Y 30.12,Z 402.613,A -85,B 0,C 180,E1 -30586.508,E2 -30586.508} C_VEL
LIN {X 0,Y 30.824,Z 402.547,A -85,B 0,C 180,E1 -30600.001,E2 -30600.001} C_VEL
LIN {X 0,Y 30.12,Z 402.6,A -85,B 0,C 180,E1 -30610.355,E2 -30610.355} C_VEL
LIN {X 0,Y 29.579,Z 402.665,A -85,B 0,C 180,E1 -30617.683,E2 -30617.683} C_VEL
LIN {X 0,Y 28.201,Z 402.794,A -85,B 0,C 180,E1 -30626.968,E2 -30626.968} C_VEL
LIN {X 0,Y 25.96,Z 402.967,A -85,B 0,C 180,E1 -30640.966,E2 -30640.966} C_VEL
LIN {X 0,Y 25.576,Z 402.979,A -85,B 0,C 180,E1 -30674.481,E2 -30674.481} C_VEL
LIN {X 0,Y 26.456,Z 402.905,A -85,B 0,C 180,E1 -30678.723,E2 -30678.723} C_VEL
LIN {X 0,Y 28.231,Z 402.791,A -85,B 0,C 180,E1 -30684.761,E2 -30684.761} C_VEL
LIN {X 0,Y 29.958,Z 410.723,A -85,B 0,C 180,E1 -30687.291,E2 -30687.291} C_VEL
LIN {X 0,Y 34.388,Z 437.273,A -85,B 0,C 180,E1 -30696.933,E2 -30696.933} C_VEL
LIN {X 0,Y 38.464,Z 457.09,A -85,B 0,C 180,E1 -30702.209,E2 -30702.209} C_VEL
LIN {X 0,Y 45.533,Z 496.535,A -85,B 0,C 180,E1 -30715.74,E2 -30715.74} C_VEL
LIN {X 0,Y 48.963,Z 509.329,A -85,B 0,C 180,E1 -30721.365,E2 -30721.365} C_VEL
LIN {X 0,Y 52.866,Z 519.825,A -85,B 0,C 180,E1 -30726.738,E2 -30726.738} C_VEL
LIN {X 0,Y 54.16,Z 522.665,A -85,B 0,C 180,E1 -30728.292,E2 -30728.292} C_VEL
LIN {X 0,Y 54.391,Z 523.256,A -85,B 0,C 180,E1 -30729.169,E2 -30729.169} C_VEL
LIN {X 0,Y 49.788,Z 513.707,A -85,B 0,C 180,E1 -30736.515,E2 -30736.515} C_VEL
LIN {X 0,Y 46.044,Z 502.644,A -85,B 0,C 180,E1 -30743.48,E2 -30743.48} C_VEL
LIN {X 0,Y 42.991,Z 489.127,A -85,B 0,C 180,E1 -30750.63,E2 -30750.63} C_VEL
LIN {X 0,Y 40.582,Z 474.523,A -85,B 0,C 180,E1 -30756.855,E2 -30756.855} C_VEL
LIN {X 0,Y 36.933,Z 451.494,A -85,B 0,C 180,E1 -30765.78,E2 -30765.78} C_VEL
LIN {X 0,Y 33.414,Z 423.149,A -85,B 0,C 180,E1 -30777.795,E2 -30777.795} C_VEL
LIN {X 0,Y 28.408,Z 405.786,A -85,B 0,C 180,E1 -30780.826,E2 -30780.826} C_VEL
LIN {X 0,Y 27.602,Z 402.849,A -85,B 0,C 180,E1 -30781.759,E2 -30781.759} C_VEL
LIN {X 0,Y 23.253,Z 403.051,A -85,B 0,C 180,E1 -30804.895,E2 -30804.895} C_VEL
LIN {X 0,Y 22.423,Z 403.077,A -85,B 0,C 180,E1 -30818.817,E2 -30818.817} C_VEL
LIN {X 0,Y 22.218,Z 403.084,A -85,B 0,C 180,E1 -30830.728,E2 -30830.728} C_VEL
LIN {X 0,Y 22.813,Z 403.065,A -85,B 0,C 180,E1 -30852.036,E2 -30852.036} C_VEL
LIN {X 0,Y 23.587,Z 403.042,A -85,B 0,C 180,E1 -30869.98,E2 -30869.98} C_VEL
LIN {X 0,Y 22.842,Z 403.064,A -85,B 0,C 180,E1 -30887.898,E2 -30887.898} C_VEL
LIN {X 0,Y 22.236,Z 403.083,A -85,B 0,C 180,E1 -30909.179,E2 -30909.179} C_VEL
LIN {X 0,Y 22.236,Z 403.083,A -85,B 0,C 180,E1 -30920.796,E2 -30920.796} C_VEL
LIN {X 0,Y 22.837,Z 403.064,A -85,B 0,C 180,E1 -30942.079,E2 -30942.079} C_VEL
LIN {X 0,Y 23.591,Z 403.042,A -85,B 0,C 180,E1 -30960.002,E2 -30960.002} C_VEL
LIN {X 0,Y 22.821,Z 403.065,A -85,B 0,C 180,E1 -30977.939,E2 -30977.939} C_VEL
LIN {X 0,Y 22.311,Z 403.081,A -85,B 0,C 180,E1 -30999.053,E2 -30999.053} C_VEL
LIN {X 0,Y 22.786,Z 403.066,A -85,B 0,C 180,E1 -31011.939,E2 -31011.939} C_VEL
LIN {X 0,Y 26.456,Z 402.905,A -85,B 0,C 180,E1 -31038.723,E2 -31038.723} C_VEL
LIN {X 0,Y 26.989,Z 403.378,A -85,B 0,C 180,E1 -31042.756,E2 -31042.756} C_VEL
LIN {X 0,Y 26.737,Z 405.4,A -85,B 0,C 180,E1 -31048.707,E2 -31048.707} C_VEL
LIN {X 0,Y 25.427,Z 410.485,A -85,B 0,C 180,E1 -31056.631,E2 -31056.631} C_VEL
LIN {X 0,Y 25.297,Z 414.36,A -85,B 0,C 180,E1 -31060.5,E2 -31060.5} C_VEL
LIN {X 0,Y 26.091,Z 420.031,A -85,B 0,C 180,E1 -31063.257,E2 -31063.257} C_VEL
LIN {X 0,Y 29.092,Z 431.47,A -85,B 0,C 180,E1 -31065.785,E2 -31065.785} C_VEL
LIN {X 0,Y 34.906,Z 456.661,A -85,B 0,C 180,E1 -31071.805,E2 -31071.805} C_VEL
LIN {X 0,Y 43.223,Z 494.792,A -85,B 0,C 180,E1 -31084.135,E2 -31084.135} C_VEL
LIN {X 0,Y 46.972,Z 506.892,A -85,B 0,C 180,E1 -31089.005,E2 -31089.005} C_VEL
LIN {X 0,Y 47.514,Z 508.351,A -85,B 0,C 180,E1 -31089.619,E2 -31089.619} C_VEL
LIN {X 0,Y 46.883,Z 506.922,A -85,B 0,C 180,E1 -31091.449,E2 -31091.449} C_VEL
LIN {X 0,Y 43.538,Z 497.509,A -85,B 0,C 180,E1 -31096.681,E2 -31096.681} C_VEL
LIN {X 0,Y 40.322,Z 484.788,A -85,B 0,C 180,E1 -31102.824,E2 -31102.824} C_VEL
LIN {X 0,Y 36.739,Z 467.976,A -85,B 0,C 180,E1 -31109.459,E2 -31109.459} C_VEL
LIN {X 0,Y 29.958,Z 431.935,A -85,B 0,C 180,E1 -31123.858,E2 -31123.858} C_VEL
LIN {X 0,Y 28.63,Z 423.255,A -85,B 0,C 180,E1 -31127.896,E2 -31127.896} C_VEL
LIN {X 0,Y 23.677,Z 406.618,A -85,B 0,C 180,E1 -31129.316,E2 -31129.316} C_VEL
LIN {X 0,Y 22.623,Z 403.071,A -85,B 0,C 180,E1 -31130.235,E2 -31130.235} C_VEL
LIN {X 0,Y 15.762,Z 403.178,A -85,B 0,C 180,E1 -31166.838,E2 -31166.838} C_VEL
LIN {X 0,Y 15.28,Z 403.178,A -85,B 0,C 180,E1 -31206.901,E2 -31206.901} C_VEL
LIN {X 0,Y 16.255,Z 403.178,A -85,B 0,C 180,E1 -31229.971,E2 -31229.971} C_VEL
LIN {X 0,Y 15.297,Z 403.178,A -85,B 0,C 180,E1 -31253.243,E2 -31253.243} C_VEL
LIN {X 0,Y 15.129,Z 403.178,A -85,B 0,C 180,E1 -31257.646,E2 -31257.646} C_VEL
LIN {X 0,Y 15.126,Z 403.178,A -85,B 0,C 180,E1 -31292.318,E2 -31292.318} C_VEL
LIN {X 0,Y 15.293,Z 403.178,A -85,B 0,C 180,E1 -31296.716,E2 -31296.716} C_VEL
LIN {X 0,Y 16.261,Z 403.178,A -85,B 0,C 180,E1 -31320.003,E2 -31320.003} C_VEL
LIN {X 0,Y 15.295,Z 403.178,A -85,B 0,C 180,E1 -31343.301,E2 -31343.301} C_VEL
LIN {X 0,Y 16.423,Z 403.178,A -85,B 0,C 180,E1 -31384.695,E2 -31384.695} C_VEL
LIN {X 0,Y 23.214,Z 403.189,A -85,B 0,C 180,E1 -31415.958,E2 -31415.958} C_VEL
LIN {X 0,Y 25.157,Z 411.421,A -85,B 0,C 180,E1 -31418.301,E2 -31418.301} C_VEL
LIN {X 0,Y 29.092,Z 431.47,A -85,B 0,C 180,E1 -31425.785,E2 -31425.785} C_VEL
LIN {X 0,Y 30.078,Z 437.147,A -85,B 0,C 180,E1 -31428.326,E2 -31428.326} C_VEL
LIN {X 0,Y 31.168,Z 446.308,A -85,B 0,C 180,E1 -31435.056,E2 -31435.056} C_VEL
LIN {X 0,Y 32.946,Z 457.276,A -85,B 0,C 180,E1 -31443.073,E2 -31443.073} C_VEL
LIN {X 0,Y 33.787,Z 461.042,A -85,B 0,C 180,E1 -31444.771,E2 -31444.771} C_VEL
LIN {X 0,Y 40.118,Z 486.015,A -85,B 0,C 180,E1 -31451.863,E2 -31451.863} C_VEL
LIN {X 0,Y 36.519,Z 472.557,A -85,B 0,C 180,E1 -31456.715,E2 -31456.715} C_VEL
LIN {X 0,Y 31.004,Z 450.18,A -85,B 0,C 180,E1 -31463.987,E2 -31463.987} C_VEL
LIN {X 0,Y 25.232,Z 423.721,A -85,B 0,C 180,E1 -31474.559,E2 -31474.559} C_VEL
LIN {X 0,Y 20.137,Z 406.409,A -85,B 0,C 180,E1 -31472.903,E2 -31472.903} C_VEL
LIN {X 0,Y 19.106,Z 403.175,A -85,B 0,C 180,E1 -31473.168,E2 -31473.168} C_VEL
LIN {X 0,Y 10.572,Z 403.178,A -85,B 0,C 180,E1 -31499.996,E2 -31499.996} C_VEL
LIN {X 0,Y 8.044,Z 403.178,A -85,B 0,C 180,E1 -31528.987,E2 -31528.987} C_VEL
LIN {X 0,Y 7.842,Z 403.178,A -85,B 0,C 180,E1 -31563.648,E2 -31563.648} C_VEL
LIN {X 0,Y 8.692,Z 403.178,A -85,B 0,C 180,E1 -31589.946,E2 -31589.946} C_VEL
LIN {X 0,Y 7.789,Z 403.178,A -85,B 0,C 180,E1 -31615.544,E2 -31615.544} C_VEL
LIN {X 0,Y 7.785,Z 403.178,A -85,B 0,C 180,E1 -31654.38,E2 -31654.38} C_VEL
LIN {X 0,Y 8.701,Z 403.178,A -85,B 0,C 180,E1 -31680.005,E2 -31680.005} C_VEL
LIN {X 0,Y 7.927,Z 403.178,A -85,B 0,C 180,E1 -31707.678,E2 -31707.678} C_VEL
LIN {X 0,Y 8.296,Z 403.178,A -85,B 0,C 180,E1 -31737.909,E2 -31737.909} C_VEL
LIN {X 0,Y 14.335,Z 403.178,A -85,B 0,C 180,E1 -31781.312,E2 -31781.312} C_VEL
LIN {X 0,Y 19.56,Z 403.349,A -85,B 0,C 180,E1 -31792.359,E2 -31792.359} C_VEL
LIN {X 0,Y 21.666,Z 411.45,A -85,B 0,C 180,E1 -31793.508,E2 -31793.508} C_VEL
LIN {X 0,Y 27.602,Z 436.397,A -85,B 0,C 180,E1 -31800.205,E2 -31800.205} C_VEL
LIN {X 0,Y 32.669,Z 456.307,A -85,B 0,C 180,E1 -31803.286,E2 -31803.286} C_VEL
LIN {X 0,Y 33.787,Z 461.042,A -85,B 0,C 180,E1 -31804.771,E2 -31804.771} C_VEL
LIN {X 0,Y 33.632,Z 460.931,A -85,B 0,C 180,E1 -31806.168,E2 -31806.168} C_VEL
LIN {X 0,Y 32.876,Z 458.745,A -85,B 0,C 180,E1 -31808.838,E2 -31808.838} C_VEL
LIN {X 0,Y 31.217,Z 452.935,A -85,B 0,C 180,E1 -31812.321,E2 -31812.321} C_VEL
LIN {X 0,Y 28.676,Z 443.393,A -85,B 0,C 180,E1 -31815.354,E2 -31815.354} C_VEL
LIN {X 0,Y 26.702,Z 435.819,A -85,B 0,C 180,E1 -31817.322,E2 -31817.322} C_VEL
LIN {X 0,Y 24.719,Z 428.211,A -85,B 0,C 180,E1 -31818.189,E2 -31818.189} C_VEL
LIN {X 0,Y 22.697,Z 420.613,A -85,B 0,C 180,E1 -31816.876,E2 -31816.876} C_VEL
LIN {X 0,Y 19.835,Z 409.763,A -85,B 0,C 180,E1 -31813.316,E2 -31813.316} C_VEL
LIN {X 0,Y 19.858,Z 409.826,A -85,B 0,C 180,E1 -31812.312,E2 -31812.312} C_VEL
LIN {X 0,Y 25.232,Z 430.436,A -85,B 0,C 180,E1 -31814.894,E2 -31814.894} C_VEL
LIN {X 0,Y 25.235,Z 430.404,A -85,B 0,C 180,E1 -31815.87,E2 -31815.87} C_VEL
LIN {X 0,Y 23.555,Z 423.791,A -85,B 0,C 180,E1 -31817.937,E2 -31817.937} C_VEL
LIN {X 0,Y 22.697,Z 420.613,A -85,B 0,C 180,E1 -31816.876,E2 -31816.876} C_VEL
LIN {X 0,Y 21.325,Z 417.109,A -85,B 0,C 180,E1 -31816.128,E2 -31816.128} C_VEL
LIN {X 0,Y 18.107,Z 412.41,A -85,B 0,C 180,E1 -31816.919,E2 -31816.919} C_VEL
LIN {X 0,Y 13.954,Z 408.492,A -85,B 0,C 180,E1 -31819.587,E2 -31819.587} C_VEL
LIN {X 0,Y 9.186,Z 405.491,A -85,B 0,C 180,E1 -31824.238,E2 -31824.238} C_VEL
LIN {X 0,Y 5.737,Z 404.083,A -85,B 0,C 180,E1 -31829.163,E2 -31829.163} C_VEL
LIN {X 0,Y 1.239,Z 403.207,A -85,B 0,C 180,E1 -31847.728,E2 -31847.728} C_VEL
LIN {X 0,Y 0.434,Z 403.178,A -85,B 0,C 180,E1 -31885.22,E2 -31885.22} C_VEL
LIN {X 0,Y 0.383,Z 403.178,A -85,B 0,C 180,E1 -31948.783,E2 -31948.783} C_VEL
LIN {X 0,Y 0.375,Z 403.178,A -85,B 0,C 180,E1 -32040.12,E2 -32040.12} C_VEL
LIN {X 0,Y 1.148,Z 403.178,A -85,B 0,C 180,E1 -32130.406,E2 -32130.406} C_VEL
LIN {X 0,Y 10.922,Z 403.178,A -85,B 0,C 180,E1 -32170.108,E2 -32170.108} C_VEL
LIN {X 0,Y 9.91,Z 403.178,A -85,B 0,C 180,E1 -32174.828,E2 -32174.828} C_VEL
LIN {X 0,Y 0.434,Z 403.178,A -85,B 0,C 180,E1 -32245.22,E2 -32245.22} C_VEL
LIN {X 0,Y 1.77,Z 405.178,A -85,B 0,C 180,E1 -32361.522,E2 -32361.522} C_VEL
LIN {X 0,Y 1.77,Z 600,A -85,B 0,C 180,E1 -32361.522,E2 -32361.522} C_VEL
LIN {X 0,Y 1.77,Z 600,A -85,B 0,C 180,E1 -32361.522,E2 -32361.522}

QRS_NEXT_CUT()

QRS_NEXT()
QRS_HOME()

END
